(* Logix 5000 project; controller ktclab11 vendor 1 type 14 code 150 rev 30.11; software revision 30.00 *)

TASK MainTask (continuous, watchdog 500 ms) : MainProgram

MODULES
   Local : vendor 1 type 14 code 150 (Compact 0, rev 30.11)
      Counters : Embedded (Compact 3, rev 1.1, Output RPI 20 ms)
      Discrete_IO : Embedded (Compact 1, rev 3.1, Output RPI 20 ms)
      Analog_IO : Embedded (Compact 2, rev 1.1, Output RPI 80 ms)
END_MODULES

PROGRAM MainProgram   (* main routine MainRoutine *)
VAR
   current : DINT := 20605;
   PL1 : ALIAS FOR Local:1:O.Data.1;   // OVER FLOW LIGHT
   SCALED : REAL := 20.006306;
   SLOPE : REAL := 18.58538;
   SLOPE2 : REAL := 223.02466;
   TEMP : REAL := 212.07578;
END_VAR

ROUTINE MainRoutine   (* ladder *)
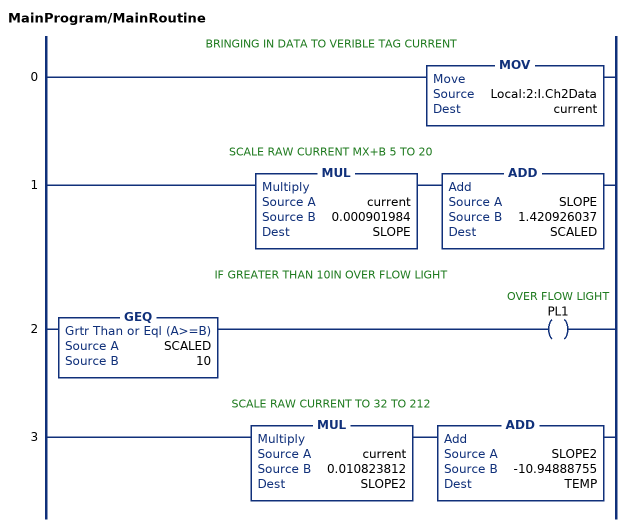
   // BRINGING IN DATA TO VERIBLE TAG CURRENT
   0: MOV(Local:2:I.Ch2Data,current);
   // SCALE RAW CURRENT MX+B 5 TO 20
   1: MUL(current,0.000901984,SLOPE)ADD(SLOPE,1.420926037,SCALED);
   // IF GREATER THAN 10IN OVER FLOW LIGHT
   2: GEQ(SCALED,10)OTE(PL1);
   // SCALE RAW CURRENT TO 32 TO 212
   3: MUL(current,0.010823812,SLOPE2)ADD(SLOPE2,-10.94888755,TEMP);
END_ROUTINE
END_PROGRAM
